// TIA Portal V18 export
FUNCTION "Motor control Function FC" : Void   // FC2, LAD
{ S7_Optimized_Access := 'TRUE' }
VERSION : 0.1
// stored: AutoNumber true, IsIECCheckEnabled false, SetENOAutomatically false, UDAEnableTagReadback false
   VAR_INPUT
      Start : Bool;   // Input to start motor
      Stop : Bool;   // input to stop motor
      "CB feedback" : Bool;
   END_VAR
   VAR_OUTPUT
      "Motor contactor" : Bool;   // Start motor contactor
   END_VAR
BEGIN

REGION Network 1: Start motor contactor
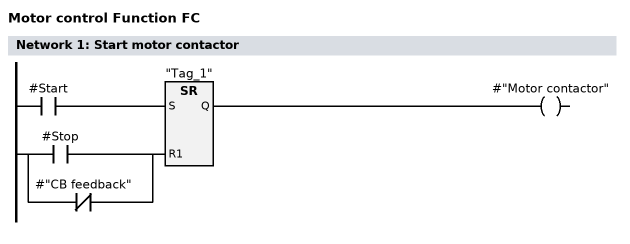
   RUNG wire#powerrail
      Contact( #Start )
      S_SR(operand := "Tag_1", r1 := wire#w1)
      Coil( #"Motor contactor" )
   END_RUNG
   RUNG wire#powerrail
      Contact( #Stop )
   END_RUNG wire#w1
   RUNG wire#powerrail
      I_Contact( #"CB feedback" )
   END_RUNG wire#w1
   // the same network as SCL:
   IF #Start THEN
       "Tag_1" := TRUE;   // SR flip-flop
   END_IF;
   IF #Stop OR NOT #"CB feedback" THEN "Tag_1" := FALSE; END_IF;
   #"Motor contactor" := "Tag_1";
END_REGION
END_FUNCTION
